(* PLC project  *)

CONFIGURATION Empty_Module_6
END_CONFIGURATION
